///EL2002 | 2-channel digital output terminal 24 V DC, 0.5 A
FUNCTION_BLOCK EL2002

VAR_INPUT
	En: BOOL;
	bDo_1: BOOL;
	bDo_2: BOOL;
	iTerminal_ID : INT;
	ErrorSystem : POINTER TO ST_ErrorSystem;
END_VAR

VAR_OUTPUT
	EnO: BOOL;
	bError: BOOL;
END_VAR

VAR
	Channel_1_Output AT %Q*: BOOL;
	Channel_2_Output AT %Q*: BOOL;
	WcState_WcState AT %I*: BOOL;
	InfoData_State AT %I*: UINT;
	
	//FB-s
	EL2002_Error : FB_TerminalError;
END_VAR

EnO:=En;

//Error FB instance
EL2002_Error(
	En := TRUE,
	iTerminal_ID := iTerminal_ID,
	bWcState := WcState_WcState,
	uiInfoData_State := InfoData_State,
	pErrorSystem := ErrorSystem,
	bError => bError,
);

IF En THEN
	IF bError=FALSE THEN
		Channel_1_Output:=bDo_1;
		Channel_2_Output:=bDo_2;
	END_IF
END_IF

END_FUNCTION_BLOCK

(* stored: Version 1.1.0.1, ProductVersion 3.1.4022.10
   POU EL2002: Id {6345d9f9-17d1-44cc-b022-fb14daef2407}, SpecialFunc None *)
